Universal Robots PolyScope program: Put_into_box_CB3_UR5_v2.urp

Program Put_into_box_CB3_UR5_v2 (installation=default directory=/programs/default createdIn=3.0.0.0 lastSavedIn=3.8.0.61336 robotSerialNumber=2018359174)
Calibrated DH parameters: a=[0, -0.425, -0.39225, 0, 0, 0]; d=[0.089159, 0, 0, 0.10915, 0.09465, 0.0823]; alpha=[1.570796, 0, 0, 1.570796, -1.570796, 0]; deltaTheta=[0, 0, 0, 0, 0, 0]
Robot Program (runOnlyOnce=true)
  Set NoAction (payload=0 tcpAsCog=true)
  MoveJ speed 10 deg/s, acceleration 80 deg/s^2 (useActiveTCP=false)
    Waypoint Home: motionParameters(blendRadius=0); TCP in base x=-99.993 y=-190.994 z=999.647 mm, rx=0.0001 ry=-2.2213 rz=2.2213 rad; joints [0, -90, 0, -90, 0, 0] deg; flange x=0 y=-191.45 z=1001.059 mm, rx=0 ry=2.2214 rz=-2.2214 rad
    Waypoint Stop: TCP in base x=42.702 y=-26.85 z=210.371 mm, rx=0 ry=-2.2214 rz=-2.2214 rad; joints [0, 0, -162, -108, 180, 90] deg
